FUNCTION_BLOCK FB_WithFields
VAR_INPUT
	InField1 	: INT;
	InField2 	: Tc2_System.ST_CpuCoreInfo;
END_VAR
VAR_IN_OUT
	InOutField1 : TIME;
END_VAR
VAR_OUTPUT
	OutField1 	: __UXINT;
	OutField2 	: Tc2_System.E_TcMemoryArea;
END_VAR
VAR
END_VAR

END_FUNCTION_BLOCK

(* stored: Version 1.1.0.1, ProductVersion 3.1.4024.15
   POU FB_WithFields: Id {56121de7-72c4-400b-94a3-0223430bf11f}, SpecialFunc None *)
